{attribute 'GeneratedUsingTerminal: EK1122-0000-0018'}
{attribute addProperty BoxType "EK1122-0000-0018"}
{attribute addProperty Id "Term_180_EK1100Term_180_EK1100_796B778320Term_182_EK1100Term_182_EK1100_E6B2C35E20"}
{attribute addProperty CRC "708014682"}
{attribute addProperty Size "40"}
{attribute addProperty Name "Term 179 (EK1122)"}
TYPE Term_179_EK1122_2A33725A EXTENDS EK1122_1FC0878B :
STRUCT
	{attribute addProperty Name "Term 180 (EK1100)"}
	{attribute addProperty PreviousPort "Term 179 (EK1122) : D"}
	{attribute addProperty SyncUnit "default"}
	Term_180_EK1100 : Term_180_EK1100_796B7783;
	{attribute addProperty Name "Term 182 (EK1100)"}
	{attribute addProperty PreviousPort "Term 179 (EK1122) : B"}
	{attribute addProperty SyncUnit "default"}
	Term_182_EK1100 : Term_182_EK1100_E6B2C35E;
END_STRUCT
END_TYPE

(* stored: Version 1.2.0.0, ProductVersion 3.1.4024.11
   DUT Term_179_EK1122_2A33725A: Id {f5b1f4b8-83cf-0d57-3fe3-26c8d0ddea3e} *)
